Fanuc KAREL source: kt00409.KL

-- PROVISIONAL review KL for V940-1; original PC SHA256 d0073661b225acc9c19dd53e6edd8758bb2caa0530b2d90478931eddee28db26
-- Incomplete behavior may be omitted. Consult companion uncertainty JSON. Do not deploy.
PROGRAM KT00409
%NOLOCKGROUP
VAR
  B1 : BOOLEAN
  B2 : BOOLEAN
  OUT : BOOLEAN
BEGIN
  -- V9_ZERO_TABLE_METADATA_HINT layout=0001; no indexed target words; source/name/runtime held
  -- UNRESOLVED_PC offsets 5-12; opcodes 9D,23
  -- UNRESOLVED_PC offsets 17-24; opcodes 9C,23
  -- UNRESOLVED_PC offsets 29-36; opcodes 9D,23
  -- UNRESOLVED_PC offsets 41-48; opcodes 9C,23
  -- UNRESOLVED_PC offsets 53-72; opcodes 21,21,5B,23
  -- UNRESOLVED_PC offsets 77-81; opcodes 7F
END KT00409
